FUNCTION_BLOCK FB_ValveCtrl52
VAR_INPUT
	i_Interlocks		:ARRAY[1..8] OF BOOL;
	i_ProcesslocksOK	:BOOL;
	i_AutoCmdHP			:BOOL;
	i_AutoCmdWP			:BOOL;
	i_ManCmdHP			:BOOL;
	i_ManCmdWP			:BOOL;
	i_ServiceMode		:BOOL;
	i_EnableHP			:BOOL;
	i_EnableWP			:BOOL;
	i_HP				:BOOL;
	i_WP				:BOOL;
	i_Timeout			:INT;
	i_MaintLimit		:UDINT;
	i_PresetValue		:UDINT;
	i_WritePreset		:BOOL;
END_VAR
VAR_OUTPUT
	q_InterlocksOK		:BOOL;
	q_Enabled			:BOOL;
	q_CmdHP				:BOOL;
	q_CmdWP				:BOOL;
	q_Traveling			:BOOL;
	q_AtHP				:BOOL;
	q_AtWP				:BOOL;
	q_TimeoutHP			:BOOL;
	q_TimeoutWP			:BOOL;
	q_SensorsFlt		:BOOL;
	q_TotalCycles		:UDINT;
	q_MaintCycles		:UDINT;
	q_MaintenanceCall	:BOOL;
	q_State				:INT;
END_VAR
VAR
	tonTimeoutHP		:TON;
	tonTimeoutWP		:TON;
	tonSensorsFlt		:TON;
	tofDelayOutHP		:TOF;
	tofDelayOutWP		:TOF;
	bCmdHP				:BOOL;
	bCmdWP				:BOOL;
END_VAR
VAR // added by the converter: edge detectors and wires of the graphical bodies
    _w1, _w2, _w3, _w4 : BOOL;
    _rt1, _rt2 : R_TRIG;
END_VAR

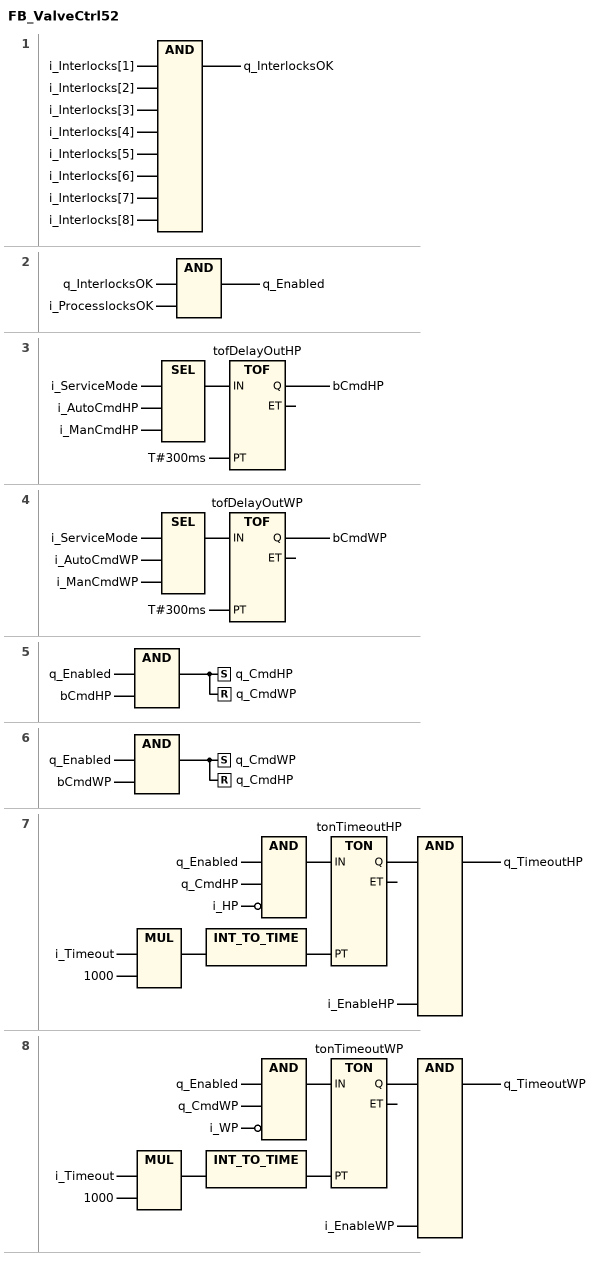
// NETWORK 1
q_InterlocksOK := i_Interlocks[1] AND i_Interlocks[2] AND i_Interlocks[3] AND i_Interlocks[4] AND i_Interlocks[5] AND i_Interlocks[6] AND i_Interlocks[7] AND i_Interlocks[8];

// NETWORK 2
q_Enabled := q_InterlocksOK AND i_ProcesslocksOK;

// NETWORK 3
tofDelayOutHP(IN := SEL(i_ServiceMode, i_AutoCmdHP, i_ManCmdHP), PT := T#300ms); // TOF
bCmdHP := tofDelayOutHP.Q;

// NETWORK 4
tofDelayOutWP(IN := SEL(i_ServiceMode, i_AutoCmdWP, i_ManCmdWP), PT := T#300ms); // TOF
bCmdWP := tofDelayOutWP.Q;

// NETWORK 5
_w1 := q_Enabled AND bCmdHP;
q_CmdHP S= _w1;
q_CmdWP R= _w1;

// NETWORK 6
_w2 := q_Enabled AND bCmdWP;
q_CmdWP S= _w2;
q_CmdHP R= _w2;

// NETWORK 7
tonTimeoutHP(IN := q_Enabled AND q_CmdHP AND NOT i_HP, PT := INT_TO_TIME(i_Timeout * 1000)); // TON
q_TimeoutHP := tonTimeoutHP.Q AND i_EnableHP;

// NETWORK 8
tonTimeoutWP(IN := q_Enabled AND q_CmdWP AND NOT i_WP, PT := INT_TO_TIME(i_Timeout * 1000)); // TON
q_TimeoutWP := tonTimeoutWP.Q AND i_EnableWP;

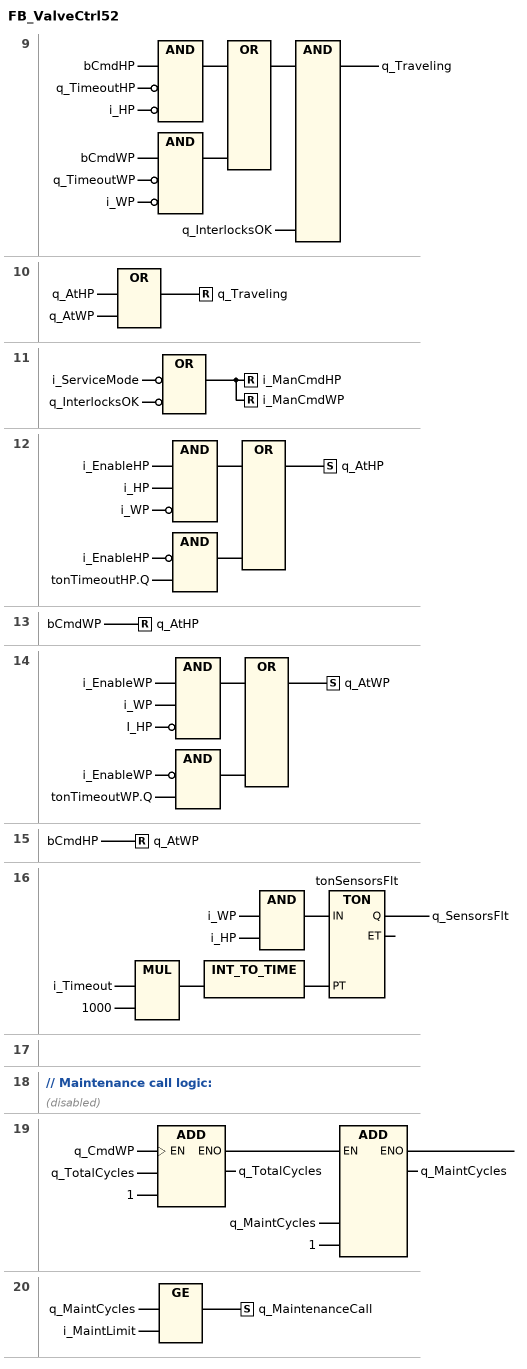
// NETWORK 9
q_Traveling := (bCmdHP AND NOT q_TimeoutHP AND NOT i_HP OR bCmdWP AND NOT q_TimeoutWP AND NOT i_WP) AND q_InterlocksOK;

// NETWORK 10
q_Traveling R= q_AtHP OR q_AtWP;

// NETWORK 11
_w3 := NOT i_ServiceMode OR NOT q_InterlocksOK;
i_ManCmdHP R= _w3;
i_ManCmdWP R= _w3;

// NETWORK 12
q_AtHP S= i_EnableHP AND i_HP AND NOT i_WP OR NOT i_EnableHP AND tonTimeoutHP.Q;

// NETWORK 13
q_AtHP R= bCmdWP;

// NETWORK 14
q_AtWP S= i_EnableWP AND i_WP AND NOT I_HP OR NOT i_EnableWP AND tonTimeoutWP.Q;

// NETWORK 15
q_AtWP R= bCmdHP;

// NETWORK 16
tonSensorsFlt(IN := i_WP AND i_HP, PT := INT_TO_TIME(i_Timeout * 1000)); // TON
q_SensorsFlt := tonSensorsFlt.Q;

// NETWORK 17

// NETWORK 18 (disabled)
// label: // Maintenance call logic

// NETWORK 19
_rt1(CLK := q_CmdWP);
_w4 := _rt1.Q;
IF _w4 THEN q_TotalCycles := q_TotalCycles + 1; END_IF
IF _w4 THEN q_MaintCycles := q_MaintCycles + 1; END_IF

// NETWORK 20
q_MaintenanceCall S= q_MaintCycles >= i_MaintLimit;

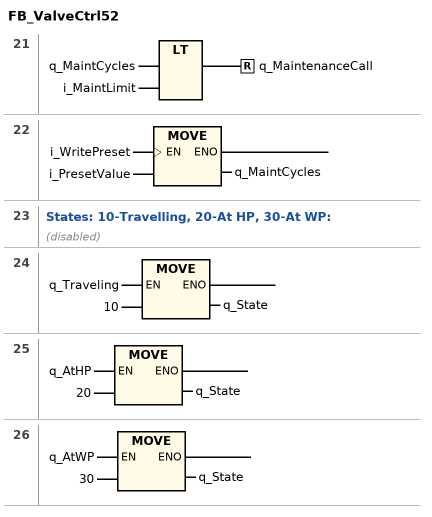
// NETWORK 21
q_MaintenanceCall R= q_MaintCycles < i_MaintLimit;

// NETWORK 22
_rt2(CLK := i_WritePreset);
IF _rt2.Q THEN q_MaintCycles := i_PresetValue; END_IF

// NETWORK 23 (disabled)
// label: States: 10-Travelling, 20-At HP, 30-At WP

// NETWORK 24
IF q_Traveling THEN q_State := 10; END_IF

// NETWORK 25
IF q_AtHP THEN q_State := 20; END_IF

// NETWORK 26
IF q_AtWP THEN q_State := 30; END_IF

END_FUNCTION_BLOCK

(* stored: Version 1.1.0.1, ProductVersion 3.1.4024.12
   POU FB_ValveCtrl52: Id {ac83a2a4-9cc5-4088-bbdb-9dc88fe075c9}, SpecialFunc None *)
